% RSLogix 500 project ONE BUTTON LATCH-UNLATCH_BAK005.RSS, saved by version 10.00.00.00 %
PROJECT "UNTITLED"    % processor: Bul.1763 MicroLogix 1100 Series B %

PROGRAM FILES
  LAD 2   5 rungs

DATA FILES
  O0 OUTPUT  4 elements
  I1 INPUT  6 elements
  S2 STATUS  66 elements
  B3 BINARY  2 elements
  T4 TIMER  1 elements
  C5 COUNTER  1 elements
  R6 CONTROL  1 elements
  N7 INTEGER  1 elements
  F8 FLOAT  1 elements

LADDER 2
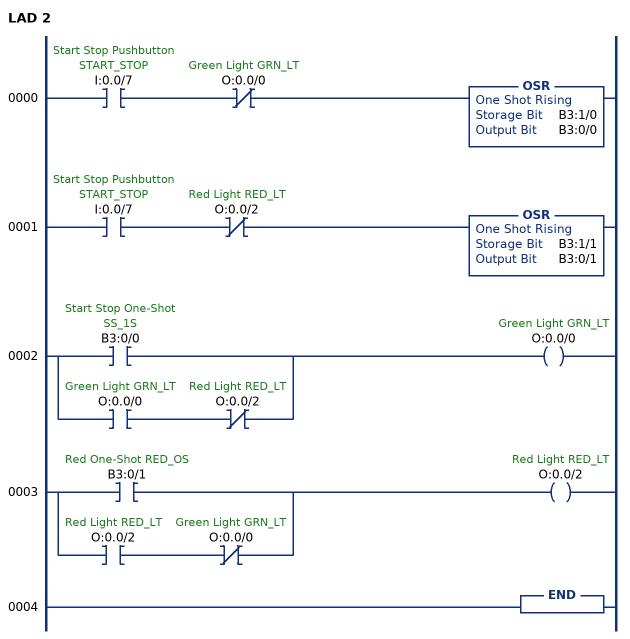
% Rung: 0 %
SOR XIC I:0.0/7 XIO O:0.0/0 OSR B3:1/0 B3:0/0 EOR
%   I:0.0/7  START_STOP  "Start Stop Pushbutton" %
%   O:0.0/0  GRN_LT  "Green Light" %
%   B3:0/0  SS_1S  "Start Stop One-Shot" %
% Rung: 1 %
SOR XIC I:0.0/7 XIO O:0.0/2 OSR B3:1/1 B3:0/1 EOR
%   I:0.0/7  START_STOP  "Start Stop Pushbutton" %
%   O:0.0/2  RED_LT  "Red Light" %
%   B3:0/1  RED_OS  "Red One-Shot" %
% Rung: 2 %
SOR BST XIC B3:0/0 NXB XIC O:0.0/0 XIO O:0.0/2 BND OTE O:0.0/0 EOR
%   B3:0/0  SS_1S  "Start Stop One-Shot" %
%   O:0.0/0  GRN_LT  "Green Light" %
%   O:0.0/2  RED_LT  "Red Light" %
% Rung: 3 %
SOR BST XIC B3:0/1 NXB XIC O:0.0/2 XIO O:0.0/0 BND OTE O:0.0/2 EOR
%   B3:0/1  RED_OS  "Red One-Shot" %
%   O:0.0/2  RED_LT  "Red Light" %
%   O:0.0/0  GRN_LT  "Green Light" %
% Rung: 4 %
SOR END EOR

OTHER DOCUMENTED ADDRESSES
  I:0.0/1  MS1_STAT  "Motor Status"
  O:0.0/4  MTR_STR  "Motor Starter"
